FUNCTION_BLOCK FB_MotionRef
VAR_INPUT
	fAmplitude : LREAL;
	fFrequency : LREAL;
	fInitialPos : LREAL;
	fCurrentPos : LREAL;
	nMotionMode : INT;
	fMotionTimer 	: LREAL;           // For selve rampen
END_VAR
VAR_OUTPUT
	fXDotRef : LREAL;
	fXRef : LREAL;
	fWantedFlow : LREAL;
END_VAR
VAR
	fPI : LREAL := 3.1415;
	fMean : LREAL;
	
	arrBounduary 	: ARRAY[0..1] OF LREAL := [G_Parameter.fPistonStroke * 0.1, G_Parameter.fPistonStroke * 0.9]; // Min, Max [m]
	fRampTime 	 	: LREAL := 15.0; // [s]
 	fTolerance   	: REAL := 0.005;  // ±5 mm
  	
END_VAR




CASE nMotionMode OF
	0:	// Sine
	
		fMean := fAmplitude + fInitialPos; 
		fXRef := fMean - fAmplitude * COS(2*fPI * fFrequency * fMotionTimer);
		fXDotRef := 2 * fPI *fFrequency * fAmplitude * SIN(2*fPI * fFrequency * fMotionTimer); 
		
	1:	// Ramp


		IF fMotionTimer <= fRampTime THEN
			fXDotRef := (arrBounduary[1] - arrBounduary[0]) / fRampTime;
			fXRef := arrBounduary[0] + fXDotRef * fMotionTimer;
		ELSIF fMotionTimer <= fRampTime * (4.0/3.0) THEN
			fXRef := arrBounduary[1];
			fXDotRef := 0.0;
		ELSIF fMotionTimer <= (2.0 + 1.0/3.0) * fRampTime AND fMotionTimer > fRampTime * (4.0/3.0) THEN
			fXDotRef := (arrBounduary[0] - arrBounduary[1]) / fRampTime;
			fXRef := arrBounduary[1] + fXDotRef * (fMotionTimer - (4.0/3.0) * fRampTime);
		ELSIF fMotionTimer > (2.0 + 1.0/3.0) * fRampTime THEN
			fXDotRef := 0.0;
			fXRef := arrBounduary[0];
		END_IF
END_CASE

IF fXDotRef > 0.0 THEN
	fWantedFlow := fXDotRef * G_Parameter.fAreaUp*6E4;
ELSIF fXDotRef < 0.0 THEN
	fWantedFlow := fXDotRef * G_Parameter.fAreaDown*6E4;
ELSE
	fWantedFlow := 0.0;
END_IF

END_FUNCTION_BLOCK

(* stored: Version 1.1.0.1, ProductVersion 3.1.4024.12
   POU FB_MotionRef: Id {354b3a34-d392-4f87-a4eb-f033618b096f}, SpecialFunc None *)
